// TIA Portal V20 program export: 3 tag tables, 23 data types, 15 data blocks, 37 code blocks (in call order from the OBs), 16 instance data blocks

VAR_GLOBAL   // PLC tag table "IO"
   "I_IN1_EXT+SGV" AT %I0.0 : Bool;   // communication spare (not used)
   "I_IN2_EXT+SGV" AT %I0.1 : Bool;   // communication spare (not used)
   "I_IN3_EXT+SGV" AT %I0.2 : Bool;   // communication spare (not used)
   "I_0E1+SGV" AT %I0.3 : Bool;   // air conditioner 1 scannerhousing visual measurement (1=ok)
   "I_0E2+SGX" AT %I0.4 : Bool;   // air conditioner scannerhousing x-ray measurement (1=ok)
   "I_0F1.1+SGV" AT %I0.5 : Bool;   // monitoring circuit breaker supply 24V ( -0F1.1)
   "I_0SH1+SSTR" AT %I0.6 : Bool;   // cooling fan / air conditioner off (cleaning filter)
   "I_14SB0+HMI" AT %I0.7 : Bool;   // emergency stop Goldeneye HMI
   "I_14SB1+HMI" AT %I1.0 : Bool;   // scanner release Goldeneye HMI
   "I_8S1.T_in" AT %I1.1 : Bool;   // adjustment top limit switch innermost position
   "I_8S2.T_out" AT %I1.2 : Bool;   // adjustment top limit switch outermost position
   "I_8S1.L_in" AT %I1.3 : Bool;   // adjustment left limit switch innermost position
   "I_8S2.L_out" AT %I1.4 : Bool;   // adjustment left limit switch outermost position
   "I_8S1.R_in" AT %I1.5 : Bool;   // adjustment right limit switch innermost position
   "I_8S2.R_out" AT %I1.6 : Bool;   // adjustment right limit switch outermost position
   "I_8S1.B_left" AT %I2.0 : Bool;   // adjustment scannerhousing limit switch left position
   "I_8S2.B_right" AT %I2.1 : Bool;   // adjustment scannerhousing limit switch right position
   "I_1BTR2+SGX" AT %I2.2 : Bool;   // light barrier in scannerhousing x-ray measurement
   "O_14VK1+SGV" AT %Q0.0 : Bool;   // safety loops scanner internal ok
   "O_14VK2+SGV" AT %Q0.1 : Bool;   // setting mode active
   "O_0VK1+SGV" AT %Q0.2 : Bool;   // scanner ready
   "O_0VK2+SGV" AT %Q0.3 : Bool;   // scanner error
   "O_0VK3+SGV" AT %Q0.4 : Bool;   // communication spare (not used)
   "O_0VK4+SGV" AT %Q0.5 : Bool;   // communication spare (not used)
   "O_0F1.1+SGV" AT %Q0.6 : Bool;   // acknowledge circuit breaker supply 24V
   "O_0KA0.1+SGV" AT %Q0.7 : Bool;   // air conditioner scannerhousing visual measurement off
   "O_0KA1+SGV" AT %Q1.1 : Bool;   // scanner status display
   "O_8M1.T_c" AT %Q1.2 : Bool;   // adjustment top close
   "O_8M1.T_o" AT %Q1.3 : Bool;   // adjustment top open
   "O_8M1.L_c" AT %Q1.4 : Bool;   // adjustment left close
   "O_8M1.L_o" AT %Q1.5 : Bool;   // adjustment left open
   "O_8M1.R_c" AT %Q1.6 : Bool;   // adjustment right close
   "O_8M1.R_o" AT %Q1.7 : Bool;   // adjustment right open
   "O_8M1.B_l" AT %Q2.1 : Bool;   // adjustment scannerhousing left
   "O_8M1.B_r" AT %Q2.2 : Bool;   // adjustment scannerhousing right
   "SI_NA_EXT+SGV" AT %I800.0 : Bool;   // emergency stop + area stop external
   "SI_14SB0/1+HMI" AT %I800.1 : Bool;   // emergency stop / scanner release Goldeneye HMI
   "SI_14SB1+SSTL" AT %I800.2 : Bool;   // setting mode scanner active
   "SI_14SB2+SSTL" AT %I800.3 : Bool;   // jog adjustment camera
   "SI_8U1+SGV" AT %I824.0 : Bool;   // adjustment linear drive monitoring
   "SI_14KA1+SGV" AT %I824.1 : Bool;   // area laser monitoring
   "SI_14KA2+SGV" AT %I824.2 : Bool;   // area adjustment monitoring
   "SI_14SS1.TL+SGV" AT %I808.0 : Bool;   // safety contact cover top left SGV
   "SI_14SS1.BL+SGV" AT %I808.1 : Bool;   // safety contact cover bottom left SGV
   "SI_14SS1.TR+SGV" AT %I808.2 : Bool;   // safety contact cover top right SGV
   "SI_14SS1.BR+SGV" AT %I808.3 : Bool;   // safety contact cover bottom right SGV
   "SI_14SS1.TL+SGX" AT %I816.0 : Bool;   // safety contact cover top left SGX
   "SI_14SS1.BL+SGX" AT %I816.1 : Bool;   // safety contact cover bottom left SGX
   "SI_14SS1.TR+SGX" AT %I816.2 : Bool;   // safety contact cover top right SGX
   "SI_14SS1.BR+SGX" AT %I816.3 : Bool;   // safety contact cover bottom right SGX
   "SO_14HV1+SSTL/R" AT %Q900.1 : Bool;   // setting mode scanner active
   "SO_14KA1+SGV" AT %Q900.2 : Bool;   // area laser on
   "SO_14KA2+SGV" AT %Q900.3 : Bool;   // area adjustment on
   "SO_ST.3HF+SGV" AT %Q908.0 : Bool;   // safety lamp laser on
   "SO_ST.5HF+SGV" AT %Q908.1 : Bool;   // safety lamp X-Ray on
   "SO_5AX1+SGX" AT %Q908.2 : Bool;   // area x-ray on
   "O_8KA1+SGV" AT %Q2.0 : Bool;   // adjustment linear drive reset (not used)
   "I_1BTR2+SGV" AT %I1.7 : Bool;   // light barrier in scannerhousing visual measurement
   "O_2YV1/2.B+SGV" AT %Q2.3 : Bool;   // blow-off valve SGV bottom
   "O_2YV1.L+SGV" AT %Q2.4 : Bool;   // blow-off valve SGV left
   "O_2YV1.R+SGV" AT %Q2.5 : Bool;   // blow-off valve SGV right
   "O_5YV1+SGX" AT %Q2.6 : Bool;   // blow-off valve SGX X-Ray
   "O_0KA0.2+SGV" AT %Q1.0 : Bool;   // air conditioner scannerhousing x-ray measurement off
   "SI_5AX1+SGX" AT %I824.3 : Bool;   // area x-ray monitoring
   O_spare27 AT %Q2.7 : Bool;   // output normal spare
   "I_0E1.1+SGV" AT %I2.3 : Bool;   // air conditioner 2 scannerhousing visual measurement (1=ok)
   I_spare24 AT %I2.4 : Bool;
   I_spare25 AT %I2.5 : Bool;
   I_spare26 AT %I2.6 : Bool;
   I_spare27 AT %I2.7 : Bool;
   SO_spare9083 AT %Q908.3 : Bool;
   SO_safetynew AT %Q900.0 : Bool;
   I_test AT %I5.0 : Bool;
END_VAR

VAR_GLOBAL   // PLC tag table "Standard-Variablentabelle"
   test0ibn AT %M0.4 : Bool;
   test1ibn AT %M0.5 : Bool;
   Tag_1 AT %M400.0 : Bool;
   Tag_2 AT %M400.1 : Bool;
   Tag_3 AT %M400.2 : Bool;
   Tag_4 AT %M2345.4 : Bool;
END_VAR
VAR_GLOBAL CONSTANT   // user constants
   USERDIAG_DEVICES_PER_SCREEN_UPPER_LIM : Int := 32;
   USERDIAG_SLOTS_PER_SCREEN_UPPER_LIM : Int := 31;
   USERDIAG_SLOTS_PER_DEVICE_UPPER_LIM : Int := 31;
   USERDIAG_DEVICES_PER_IO_SYSTEM_UPPER_LIM : Int := 128;
   USERDIAG_SLOTS_PER_PLC_UPPER_LIM : Int := 31;
END_VAR

VAR_GLOBAL   // PLC tag table "Standard"
   false AT %M0.0 : Bool;
   true AT %M0.1 : Bool;
   test0 AT %M0.2 : Bool;
   test1 AT %M0.3 : Bool;
   dummy AT %M0.7 : Bool;
   clockFlag10Hz AT %M1.0 : Bool;   // ClockFlag 0.1s
   clockFlag5Hz AT %M1.1 : Bool;   // ClockFlag 0.2s
   flash AT %M1.2 : Bool;   // ClockFlag 0.4s
   clockFlag2Hz AT %M1.3 : Bool;   // ClockFlag 0.5s
   blinker AT %M1.4 : Bool;   // ClockFlag 0.8s
   clockFlag1Hz AT %M1.5 : Bool;   // ClockFlag 1.0s
   "clockFlag0,625Hz" AT %M1.6 : Bool;   // ClockFlag 1.6s
   "clockFlag0,5Hz" AT %M1.7 : Bool;   // ClockFlag 2.0s
   cycleFlag AT %MB2 : Byte;
   cycleFlash AT %M2.0 : Bool;
   systemByte AT %MB3 : Byte;
   firstScan AT %M3.0 : Bool;   // cpu startup
   diagStatusUpdate AT %M3.1 : Bool;
   alwaysTRUE AT %M3.2 : Bool;
   alwaysFALSE AT %M3.3 : Bool;
   clockByte AT %MB1 : Byte;
   cycle AT %MD6 : Real;   // program cycle in ms
   "real" AT %MD10 : Real;
   "dWord" AT %MD18 : DWord;
   "dint" AT %MD14 : DInt;
   "int" AT %MW22 : Int;
   "word" AT %MW24 : Word;
   "byte" AT %MB26 : Byte;
   "bool" AT %M27.0 : Bool;
   systemClockByte AT %MB30 : Byte;
   clockTest AT %M0.6 : Bool;
   T0 AT %T0 : Timer;
   T1 AT %T1 : Timer;
   T2 AT %T2 : Timer;
   mem AT %M32.0 : LReal;
   T3 AT %T3 : Timer;
END_VAR

TYPE "TypeAxisRd"
   STRUCT
      TargetPos : DInt;   // target position [mm/10]
      CalibratePos : DInt;   // calibrated position [mm/10]
      RefPosToBoard : DInt;   // reference position to board [mm/10]
      SetCalibratePos : Bool;   // set calibrated position
      ManModeActive : Bool;   // manual mode active
      ManPlus : Bool;   // manual plus
      ManMinus : Bool;   // manual minus
      ManRefRun : Bool;   // manual reference run
   END_STRUCT;
END_TYPE

TYPE "TypeAxisSd"
   STRUCT
      ActualEncPos : DInt;   // actual encoder position [mm/10]
      ActualPos : DInt;   // actual position [mm/10]
      LimitSwitchMin : Bool;   // limit switch min active
      LimitSwitchMax : Bool;   // limit switch max active
      Err : Bool;   // error
      ErrEnc : Bool;   // error encoder
      PosOk : Bool;   // position ok
      Plus : Bool;   // moves plus
      Minus : Bool;   // moves minus
      refRun : Bool;   // reference running
      refOk : Bool;   // reference ok
      SetCalibratePosOk : Bool;   // set calibrated position ok
   END_STRUCT;
END_TYPE

TYPE "TypeCmd"
   STRUCT
      auto : Bool;   // automatic mode
      autoP : Bool;   // automatic plus
      autoM : Bool;   // automatic minus
      autoLift : Bool;   // automatic lift
      autoLower : Bool;   // automatic lower
      man : Bool;   // manual mode
      manP : Bool;   // manual plus
      manM : Bool;   // manual minus
      manLift : Bool;   // manual lift
      manLower : Bool;   // manual lower
      enable : Bool;   // release
      enPlus : Bool;   // release plus
      enMinus : Bool;   // release minus
      enLift : Bool;   // release lift
      enLower : Bool;   // release lower
      enAutoP : Bool;   // release automatic plus
      enAutoM : Bool;   // release automatic minus
      enAutoLift : Bool;   // release automatic lift
      enAutoLower : Bool;   // release automatic lower
      slow : Bool;
      lamp : Bool;   // indication lamp
      ack : Bool;   // fault acknowledge
      cycle : Bool;   // cycle start
      goToGpos : Bool;   // go to groundposition
      goToCpos : Bool;   // go to cm-position
      goToEpos : Bool;   // go to endpos
      goToWPos : Bool;   // go to wait/fly position
      inGpos : Bool;   // in groundposition
      inCpos : Bool;   // in cm-position
      inEpos : Bool;   // in endpos
      inWPos : Bool;   // in wait/fly position
      speed : Int;   // Desired speed raw in Hz or Upm
      tarSpeed : Real;   // target speed
      mmCycle : Real;   // milimeter per cycle
      gain : Real;   // gain
      ramp : Int;   // ramp
      startRamp : Int;   // start ramp
      stopRamp : Int;   // stop ramp
      gPos : Real;   // Desired value basic position [mm]
      cPos : Real;   // Desired value cm position [mm]
      ePos : Real;   // Desired value end position [mm]
      wPos : Real;   // Desired value wait/fly position [mm]
      tarMax : Real;   // target maximum
      tarMin : Real;   // target minimum
      target : Real;
      actual : Real;
   END_STRUCT;
END_TYPE

TYPE "TypeHeaderPcGld"
   STRUCT
      valid : Int;   // valid
      watchdog : Int;   // watchdog
      bit40 : Bool;
      ack : Bool;   // acknowledge
      bit42 : Bool;
      bit43 : Bool;
      bit44 : Bool;
      bit45 : Bool;
      bit46 : Bool;
      bit47 : Bool;
      word6 : Word;
      word8 : Word;
   END_STRUCT;
END_TYPE

TYPE "TypeHeaderPlc"
   STRUCT
      conActive : Bool;   // connection is established
      err : Bool;   // fault general
      errWd : Bool;   // fault watchdog
      errSd : Bool;   // fault send
      errRd : Bool;   // fault receive
      bit05 : Bool;
      bit06 : Bool;
      bit07 : Bool;
      sdBusy : Bool;   // new data is sending
      sdDone : Bool;   // new data sended
      rdBusy : Bool;   // new data is receiving
      rdDone : Bool;   // new data received
      sdOverload : Bool;   // new data could not be sent because the Cp overloaded
      statistic : Bool;   // statistic information are aviable
      bit16 : Bool;
      bit17 : Bool;
      sdState : Word;   // send state
      sdLastErrState : Word;   // send last fault state
      sdLenght : Int;   // send lenght [byte]
      sdCps : Int;   // send counter per second
      rdState : Word;   // receive state
      rdLastErrState : Word;   // receive last fault state
      rdLenght : Int;   // receive lenght [byte]
      rdCps : Int;   // receive counter per second
      in18 : Int;
   END_STRUCT;
END_TYPE

TYPE "TypeSensor"
   STRUCT
      sen : Bool;
      onDel : Bool;
      offDel : Bool;
      occ : Bool;
      occPe : Bool;
      occNe : Bool;
      off : Bool;
      full : Bool;
      free : Bool;
      empty : Bool;
      err : Bool;
      errOcc : Bool;   // fault sensor was to long occupied, maybe dirty or misaligned
      errFree : Bool;   // fault sensor was to long free, maybe dirty or misaligned
      errCycle : Bool;   // fault sensor plausibility check of cycles, after a certain amount(#errCycleVal) of trigger(#errCycleIn) the sensor had no rising or falling edge
      war : Bool;
      refMode : Bool;   // reference mode
      refRun : Bool;   // reference running
      onCntr : Real;   // counter for on delayed
      offCntr : Real;   // counter for off delayed
      occOnCntr : Real;   // on counter for occupied
      occOffCntr : Real;   // on counter for occupied
      val : Real;   // value from sensor, if ex. the sensor is read as a analog input
      occGap : Real;   // gap since last occupied
      "name" : WString[30];   // name, used for fault messages
      description : WString[90];   // description, used for fault messages
   END_STRUCT;
END_TYPE

TYPE "TypeVar"
   STRUCT
      "bool" { ExternalAccessible := 'False'; ExternalVisible := 'False'; ExternalWritable := 'False'} : Bool;
      "byte" { ExternalAccessible := 'False'; ExternalVisible := 'False'; ExternalWritable := 'False'} : Byte;
      "word" { ExternalAccessible := 'False'; ExternalVisible := 'False'; ExternalWritable := 'False'} : Word;
      "dword" { ExternalAccessible := 'False'; ExternalVisible := 'False'; ExternalWritable := 'False'} : DWord;
      "int" { ExternalAccessible := 'False'; ExternalVisible := 'False'; ExternalWritable := 'False'} : Int;
      "dint" { ExternalAccessible := 'False'; ExternalVisible := 'False'; ExternalWritable := 'False'} : DInt;
      "real" { ExternalAccessible := 'False'; ExternalVisible := 'False'; ExternalWritable := 'False'} : Real;
      s5time { ExternalAccessible := 'False'; ExternalVisible := 'False'; ExternalWritable := 'False'} : S5Time;
      "time" { ExternalAccessible := 'False'; ExternalVisible := 'False'; ExternalWritable := 'False'} : Time;
      hm1 { ExternalAccessible := 'False'; ExternalVisible := 'False'; ExternalWritable := 'False'} : Bool;
      hm2 { ExternalAccessible := 'False'; ExternalVisible := 'False'; ExternalWritable := 'False'} : Bool := false;
      hm3 { ExternalAccessible := 'False'; ExternalVisible := 'False'; ExternalWritable := 'False'} : Bool := false;
      hm4 { ExternalAccessible := 'False'; ExternalVisible := 'False'; ExternalWritable := 'False'} : Bool := false;
      hm5 { ExternalAccessible := 'False'; ExternalVisible := 'False'; ExternalWritable := 'False'} : Bool := false;
      hm6 { ExternalAccessible := 'False'; ExternalVisible := 'False'; ExternalWritable := 'False'} : Bool := false;
      hm7 { ExternalAccessible := 'False'; ExternalVisible := 'False'; ExternalWritable := 'False'} : Bool := false;
      hm8 { ExternalAccessible := 'False'; ExternalVisible := 'False'; ExternalWritable := 'False'} : Bool := false;
      hm9 { ExternalAccessible := 'False'; ExternalVisible := 'False'; ExternalWritable := 'False'} : Bool := false;
      hm10 { ExternalAccessible := 'False'; ExternalVisible := 'False'; ExternalWritable := 'False'} : Bool := false;
      hm11 { ExternalAccessible := 'False'; ExternalVisible := 'False'; ExternalWritable := 'False'} : Bool := false;
      hm12 { ExternalAccessible := 'False'; ExternalVisible := 'False'; ExternalWritable := 'False'} : Bool := false;
      hm13 { ExternalAccessible := 'False'; ExternalVisible := 'False'; ExternalWritable := 'False'} : Bool := false;
      hm14 { ExternalAccessible := 'False'; ExternalVisible := 'False'; ExternalWritable := 'False'} : Bool := false;
      hm15 { ExternalAccessible := 'False'; ExternalVisible := 'False'; ExternalWritable := 'False'} : Bool := false;
      hm16 { ExternalAccessible := 'False'; ExternalVisible := 'False'; ExternalWritable := 'False'} : Bool := false;
      fm1 { ExternalAccessible := 'False'; ExternalVisible := 'False'; ExternalWritable := 'False'} : Bool;
      fm2 { ExternalAccessible := 'False'; ExternalVisible := 'False'; ExternalWritable := 'False'} : Bool := false;
      fm3 { ExternalAccessible := 'False'; ExternalVisible := 'False'; ExternalWritable := 'False'} : Bool := false;
      fm4 { ExternalAccessible := 'False'; ExternalVisible := 'False'; ExternalWritable := 'False'} : Bool := false;
      fm5 { ExternalAccessible := 'False'; ExternalVisible := 'False'; ExternalWritable := 'False'} : Bool := false;
      fm6 { ExternalAccessible := 'False'; ExternalVisible := 'False'; ExternalWritable := 'False'} : Bool := false;
      fm7 { ExternalAccessible := 'False'; ExternalVisible := 'False'; ExternalWritable := 'False'} : Bool := false;
      fm8 { ExternalAccessible := 'False'; ExternalVisible := 'False'; ExternalWritable := 'False'} : Bool := false;
      fm9 { ExternalAccessible := 'False'; ExternalVisible := 'False'; ExternalWritable := 'False'} : Bool := false;
      fm10 { ExternalAccessible := 'False'; ExternalVisible := 'False'; ExternalWritable := 'False'} : Bool := false;
      fm11 { ExternalAccessible := 'False'; ExternalVisible := 'False'; ExternalWritable := 'False'} : Bool := false;
      fm12 { ExternalAccessible := 'False'; ExternalVisible := 'False'; ExternalWritable := 'False'} : Bool := false;
      fm13 { ExternalAccessible := 'False'; ExternalVisible := 'False'; ExternalWritable := 'False'} : Bool := false;
      fm14 { ExternalAccessible := 'False'; ExternalVisible := 'False'; ExternalWritable := 'False'} : Bool := false;
      fm15 { ExternalAccessible := 'False'; ExternalVisible := 'False'; ExternalWritable := 'False'} : Bool := false;
      fm16 { ExternalAccessible := 'False'; ExternalVisible := 'False'; ExternalWritable := 'False'} : Bool := false;
      bool1 { ExternalAccessible := 'False'; ExternalVisible := 'False'; ExternalWritable := 'False'} : Bool;
      bool2 { ExternalAccessible := 'False'; ExternalVisible := 'False'; ExternalWritable := 'False'} : Bool;
      bool3 { ExternalAccessible := 'False'; ExternalVisible := 'False'; ExternalWritable := 'False'} : Bool;
      bool4 { ExternalAccessible := 'False'; ExternalVisible := 'False'; ExternalWritable := 'False'} : Bool;
      bool5 { ExternalAccessible := 'False'; ExternalVisible := 'False'; ExternalWritable := 'False'} : Bool;
      bool6 { ExternalAccessible := 'False'; ExternalVisible := 'False'; ExternalWritable := 'False'} : Bool;
      bool7 { ExternalAccessible := 'False'; ExternalVisible := 'False'; ExternalWritable := 'False'} : Bool;
      bool8 { ExternalAccessible := 'False'; ExternalVisible := 'False'; ExternalWritable := 'False'} : Bool;
      bool9 { ExternalAccessible := 'False'; ExternalVisible := 'False'; ExternalWritable := 'False'} : Bool;
      bool10 { ExternalAccessible := 'False'; ExternalVisible := 'False'; ExternalWritable := 'False'} : Bool;
      bool11 { ExternalAccessible := 'False'; ExternalVisible := 'False'; ExternalWritable := 'False'} : Bool;
      bool12 { ExternalAccessible := 'False'; ExternalVisible := 'False'; ExternalWritable := 'False'} : Bool;
      bool13 { ExternalAccessible := 'False'; ExternalVisible := 'False'; ExternalWritable := 'False'} : Bool;
      bool14 { ExternalAccessible := 'False'; ExternalVisible := 'False'; ExternalWritable := 'False'} : Bool;
      bool15 { ExternalAccessible := 'False'; ExternalVisible := 'False'; ExternalWritable := 'False'} : Bool;
      bool16 { ExternalAccessible := 'False'; ExternalVisible := 'False'; ExternalWritable := 'False'} : Bool;
      int1 { ExternalAccessible := 'False'; ExternalVisible := 'False'; ExternalWritable := 'False'} : Int;
      int2 { ExternalAccessible := 'False'; ExternalVisible := 'False'; ExternalWritable := 'False'} : Int := 0;
      int3 { ExternalAccessible := 'False'; ExternalVisible := 'False'; ExternalWritable := 'False'} : Int := 0;
      int4 { ExternalAccessible := 'False'; ExternalVisible := 'False'; ExternalWritable := 'False'} : Int := 0;
      int5 { ExternalAccessible := 'False'; ExternalVisible := 'False'; ExternalWritable := 'False'} : Int := 0;
      int6 { ExternalAccessible := 'False'; ExternalVisible := 'False'; ExternalWritable := 'False'} : Int := 0;
      int7 { ExternalAccessible := 'False'; ExternalVisible := 'False'; ExternalWritable := 'False'} : Int := 0;
      int8 { ExternalAccessible := 'False'; ExternalVisible := 'False'; ExternalWritable := 'False'} : Int := 0;
      int9 { ExternalAccessible := 'False'; ExternalVisible := 'False'; ExternalWritable := 'False'} : Int := 0;
      int10 { ExternalAccessible := 'False'; ExternalVisible := 'False'; ExternalWritable := 'False'} : Int := 0;
      word1 { ExternalAccessible := 'False'; ExternalVisible := 'False'; ExternalWritable := 'False'} : Word;
      word2 { ExternalAccessible := 'False'; ExternalVisible := 'False'; ExternalWritable := 'False'} : Word := 16#0;
      word3 { ExternalAccessible := 'False'; ExternalVisible := 'False'; ExternalWritable := 'False'} : Word := 16#0;
      word4 { ExternalAccessible := 'False'; ExternalVisible := 'False'; ExternalWritable := 'False'} : Word := 16#0;
      word5 { ExternalAccessible := 'False'; ExternalVisible := 'False'; ExternalWritable := 'False'} : Word := 16#0;
      word6 { ExternalAccessible := 'False'; ExternalVisible := 'False'; ExternalWritable := 'False'} : Word := 16#0;
      word7 { ExternalAccessible := 'False'; ExternalVisible := 'False'; ExternalWritable := 'False'} : Word := 16#0;
      word8 { ExternalAccessible := 'False'; ExternalVisible := 'False'; ExternalWritable := 'False'} : Word := 16#0;
      word9 { ExternalAccessible := 'False'; ExternalVisible := 'False'; ExternalWritable := 'False'} : Word := 16#0;
      word10 { ExternalAccessible := 'False'; ExternalVisible := 'False'; ExternalWritable := 'False'} : Word := 16#0;
      real1 { ExternalAccessible := 'False'; ExternalVisible := 'False'; ExternalWritable := 'False'} : Real;
      real2 { ExternalAccessible := 'False'; ExternalVisible := 'False'; ExternalWritable := 'False'} : Real := 0.0;
      real3 { ExternalAccessible := 'False'; ExternalVisible := 'False'; ExternalWritable := 'False'} : Real := 0.0;
      real4 { ExternalAccessible := 'False'; ExternalVisible := 'False'; ExternalWritable := 'False'} : Real := 0.0;
      real5 { ExternalAccessible := 'False'; ExternalVisible := 'False'; ExternalWritable := 'False'} : Real := 0.0;
      real6 { ExternalAccessible := 'False'; ExternalVisible := 'False'; ExternalWritable := 'False'} : Real := 0.0;
      real7 { ExternalAccessible := 'False'; ExternalVisible := 'False'; ExternalWritable := 'False'} : Real := 0.0;
      real8 { ExternalAccessible := 'False'; ExternalVisible := 'False'; ExternalWritable := 'False'} : Real := 0.0;
      real9 { ExternalAccessible := 'False'; ExternalVisible := 'False'; ExternalWritable := 'False'} : Real := 0.0;
      real10 { ExternalAccessible := 'False'; ExternalVisible := 'False'; ExternalWritable := 'False'} : Real := 0.0;
   END_STRUCT;
END_TYPE

TYPE "UserDiag_typeActIOSystem"
TITLE = UserDiag_typeActIOSystem
   STRUCT
      actIOSystemNumber : Int := 1;   // Number of actual selected IO-system/DP-Mastersystem
      actIODeviceNumbers : Array[1.."USERDIAG_DEVICES_PER_SCREEN_UPPER_LIM"] of UInt;   // Device numbers/profibus addresses of actual selected IO-System/DP-Mastersystem
      actIODeviceState : Array[1.."USERDIAG_DEVICES_PER_SCREEN_UPPER_LIM"] of USInt;   // State of devices/slaves in actual selected IO-System/DP-Mastersystem
      actDeviceSlotsUsed : Array[0.."USERDIAG_SLOTS_PER_SCREEN_UPPER_LIM"] of Bool;   // Used slots of actual selected device/slave
      actDeviceSlotsState : Array[0.."USERDIAG_SLOTS_PER_SCREEN_UPPER_LIM"] of USInt;   // States of actual selected device/slave
   END_STRUCT;
END_TYPE

TYPE "UserDiag_typeDevice"
TITLE = UserDiag_typeDevice
   STRUCT
      hardwareId { ExternalAccessible := 'False'; ExternalVisible := 'False'; ExternalWritable := 'False'} : HW_DEVICE := 16#0000;   // Hardware identifier of the device/slave
      number { ExternalAccessible := 'False'; ExternalVisible := 'False'; ExternalWritable := 'False'} : UInt := 0;   // Profinet device number/Profibus address of the slave
      "name" { ExternalAccessible := 'False'; ExternalVisible := 'False'; ExternalWritable := 'False'} : String[50];   // Name of the device/slave
      ipAddress { ExternalAccessible := 'False'; ExternalVisible := 'False'; ExternalWritable := 'False'; S7_SetPoint := 'True'} : IP_V4;   // IP address of the device
      state { ExternalAccessible := 'False'; ExternalVisible := 'False'; ExternalWritable := 'False'} : USInt := 0;   // Status of the device/slave. 1:ok; 2:faulty, 3:lost connection, 4:disabled, 5:problem, 12:was faulty, 13:was lost, 14:was disabled, 15:problem gone
      exists { ExternalAccessible := 'False'; ExternalVisible := 'False'; ExternalWritable := 'False'} : Bool := FALSE;   // TRUE: Device/slave is existing
      configured { ExternalAccessible := 'False'; ExternalVisible := 'False'; ExternalWritable := 'False'} : Bool := FALSE;   // TRUE: Device/slave is configured
      faulty { ExternalAccessible := 'False'; ExternalVisible := 'False'; ExternalWritable := 'False'} : Bool := FALSE;   // TRUE: Device/slave is faulty
      problem { ExternalAccessible := 'False'; ExternalVisible := 'False'; ExternalWritable := 'False'} : Bool := FALSE;   // TRUE: Device/slave has a problem
      disabled { ExternalAccessible := 'False'; ExternalVisible := 'False'; ExternalWritable := 'False'} : Bool := FALSE;   // TRUE: Device/slave is disabled
      error { ExternalAccessible := 'False'; ExternalVisible := 'False'; ExternalWritable := 'False'} : Bool := FALSE;   // TRUE: Error in device/slave
      nextDevice { ExternalAccessible := 'False'; ExternalVisible := 'False'; ExternalWritable := 'False'} : Int;   // device number of next device
      actualConfiguredSlots { ExternalAccessible := 'False'; ExternalVisible := 'False'; ExternalWritable := 'False'} : Int := 0;   // Number of configured slots in the device/slave
      slots { ExternalAccessible := 'False'; ExternalVisible := 'False'; ExternalWritable := 'False'; S7_SetPoint := 'True'} : Array[0.."USERDIAG_SLOTS_PER_DEVICE_UPPER_LIM"] of "UserDiag_typeSlot";   // Slot information of a device/slave
   END_STRUCT;
END_TYPE

TYPE "UserDiag_typeDiagnostics"
TITLE = UserDiag_typeDiagnostics
   STRUCT
      subfunctionStatus : Word := 16#0000;   // Block status or error information
      instructionError : Int := 0;   // Indicates in which system function the error occurred. 1:DeviceStates PN; 2=GetName PN; 3:ModuleStates PN; 4:DeviceStates DP; 5:GetName DP; 6:ModuleStates DP
      errorIndex : Int := 0;   // The last index of the respective loop, if an error occures (relevant for IOSystemCheck FB)
   END_STRUCT;
END_TYPE

TYPE "UserDiag_typeIOSystem"
TITLE = UserDiag_typeIOSystem
   STRUCT
      hardwareId { ExternalAccessible := 'False'; ExternalVisible := 'False'; ExternalWritable := 'False'} : HW_IOSYSTEM := 16#0000;   // Hardware identifier of the IO-System/DP-Mastersystem
      number { ExternalAccessible := 'False'; ExternalVisible := 'False'; ExternalWritable := 'False'} : UInt := 0;   // IO-System/DP-Mastersystem number
      error { ExternalAccessible := 'False'; ExternalVisible := 'False'; ExternalWritable := 'False'} : Bool := FALSE;   // TRUE: Error in IO-System/DP-Mastersystem
      firstDevice { ExternalAccessible := 'False'; ExternalVisible := 'False'; ExternalWritable := 'False'} : Int := 0;   // device number (index) of first device in IO System
      lastDevice { ExternalAccessible := 'False'; ExternalVisible := 'False'; ExternalWritable := 'False'} : Int := 0;   // device number (index) of last device IO System
      actualConfiguredDevices { ExternalAccessible := 'False'; ExternalVisible := 'False'; ExternalWritable := 'False'} : Int := 0;   // Number of configured devices/slaves in IO-System/DP-Mastersystem
      devices { ExternalAccessible := 'False'; ExternalVisible := 'False'; ExternalWritable := 'False'; S7_SetPoint := 'True'} : Array[1.."USERDIAG_DEVICES_PER_IO_SYSTEM_UPPER_LIM"] of "UserDiag_typeDevice";   // Device/Slave information
   END_STRUCT;
END_TYPE

TYPE "UserDiag_typePLC"
TITLE = UserDiag_typePLC
   STRUCT
      hardwareId { ExternalAccessible := 'False'; ExternalVisible := 'False'; ExternalWritable := 'False'} : HW_DEVICE := 16#0000;   // Hardware identifier of the PLC
      error { ExternalAccessible := 'False'; ExternalVisible := 'False'; ExternalWritable := 'False'} : Bool := FALSE;   // TRUE: Error in PLC
      errorLedActive { ExternalAccessible := 'False'; ExternalVisible := 'False'; ExternalWritable := 'False'} : Bool := FALSE;   // TRUE: PLC led signals an error
      actualConfiguredSlots { ExternalAccessible := 'False'; ExternalVisible := 'False'; ExternalWritable := 'False'} : Int := 0;   // Number of configured local slots at PLC
      slots { ExternalAccessible := 'False'; ExternalVisible := 'False'; ExternalWritable := 'False'; S7_SetPoint := 'True'} : Array[0.."USERDIAG_SLOTS_PER_PLC_UPPER_LIM"] of "UserDiag_typeSlot";   // Information of the PLC slots; index = slotnumber; PLC always at slot 1
   END_STRUCT;
END_TYPE

TYPE "UserDiag_typeSlot"
TITLE = UserDiag_typeSlot
   STRUCT
      hardwareId { ExternalAccessible := 'False'; ExternalVisible := 'False'; ExternalWritable := 'False'} : HW_IO := 16#0000;   // Hardware identifier of the module which is inserted in the slot
      state { ExternalAccessible := 'False'; ExternalVisible := 'False'; ExternalWritable := 'False'} : USInt := 0;   // Status of the device/slave. 1:ok; 2:faulty, 3:lost connection, 4:disabled, 5:problem, 12:was faulty, 13:was lost, 14:was disabled, 15:problem gone
      exists { ExternalAccessible := 'False'; ExternalVisible := 'False'; ExternalWritable := 'False'} : Bool := FALSE;   // TRUE: Modul is existing
      configured { ExternalAccessible := 'False'; ExternalVisible := 'False'; ExternalWritable := 'False'} : Bool := FALSE;   // TRUE: Modul is configured
      faulty { ExternalAccessible := 'False'; ExternalVisible := 'False'; ExternalWritable := 'False'} : Bool := FALSE;   // TRUE: Modul is faulty
      problem { ExternalAccessible := 'False'; ExternalVisible := 'False'; ExternalWritable := 'False'} : Bool := FALSE;   // TRUE: Modul has a problem
      disabled { ExternalAccessible := 'False'; ExternalVisible := 'False'; ExternalWritable := 'False'} : Bool := FALSE;   // TRUE: Modul is disabled
      error { ExternalAccessible := 'False'; ExternalVisible := 'False'; ExternalWritable := 'False'} : Bool := FALSE;   // TRUE: Error in module which is inserted in the slot
   END_STRUCT;
END_TYPE

TYPE "TypeLinmotRd"
   STRUCT
      StatVar : Struct   // State Var
         SubState : Byte;   // main state
         MainState : Byte;   // sub state
      END_STRUCT;
      StatWord : Struct   // Status Word
         OperationEnabled : Bool;   // 1 = State Nr 8 or higher (copied to drive EN LED )
         SwitchOnActive : Bool;   // 1 = Control Word Bit 0
         EnableOperation : Bool;   // 1 = Control Word Bit 3
         Error : Bool;   // 1 = Error
         VoltageEnable : Bool;   // 1 = Control Word Bit 1
         QuickStop : Bool;   // 1 = Control Word Bit 2
         SwitchOnLocked : Bool;   // 1= Release with 0 of Control word bit 0 (Switch On)
         Warning : Bool;   // 1 = One or more bits in the Warn Word are set
         EventHandlerActive : Bool;   // Event Handler setup
         SpecialMotionActive : Bool;   // Special motion commands (Homing, ..) runs
         InTargetPosition : Bool;   // Actual position after motion in window
         Homed : Bool;   // Position sensor system valid
         FatalError : Bool;   // A fatal error can not be acknowledged!
         MotionActive : Bool;   // Setpoint generation (VAI, curve) active
         RangeIndicator1 : Bool;   // Defined UPID is in Range 1
         RangeIndicator2 : Bool;   // Defined UPID is in Range 2
      END_STRUCT;
      WarnWord : Struct   // Warning Word
         MotorHotSensor : Bool;
         MotorShortTimerOverload : Bool;
         MotorSupplyVoltageLow : Bool;
         MotorSupplyVoltageHigh : Bool;
         PositionLagAlways : Bool;
         Res5 : Bool;
         DriveHot : Bool;
         MotorNotHomed : Bool;
         PTC_Sensor1Hot : Bool;
         PTC_Sensor2Hot : Bool;
         Res10 : Bool;
         Res11 : Bool;
         Res12 : Bool;
         Res13 : Bool;
         InterfaceWarnFlag : Bool;
         ApplicationWarnFlag : Bool;
      END_STRUCT;
      Tarpos : DInt;   // target position
      Actpos : DInt;   // actual position
      TarCurrent : DInt;   // target current
      CfgStatWord : Int;   // config status word
      CfgId : Int;   // config index response
      CfgVal : DInt;   // config value response
   END_STRUCT;
END_TYPE

TYPE "TypeLinmotSd"
   STRUCT
      Ctrl : Struct   // control word
         SwitchOn : Bool;   // 0 = A-Stop, -> Current = 0, power switches disabled
         VoltageEnable : Bool;   // 0 = Power switches disabled without microcontroller action
         QuickStop : Bool;   // 0 = Quick Stop -> Current = 0 -> H-Bridges disabled
         EnableOperation : Bool;   // Position controller active Motion Commands enabled
         Abort : Bool;   // 0 = Quick Stop position control rests active, motion
         Freeze : Bool;   // 0 = Quick Stop position control rests active, Target position
         GoToPosition : Bool;   // 1 = Go to fixed parameterized Position. Wait for release of signal
         ErrorAcknoledge : Bool;   // 1 = Rising edge of signal acknowledges error
         JogMovePlus : Bool;   // 1 = Jog Move +
         JogMoveMinus : Bool;   // 1 = Jog Move -
         SpecialMove : Bool;   // 1 = Special Mode
         Home : Bool;   // 1 = At startup bit 11 Status word is cleared, until procedure
         ClearanceCheck : Bool;   // 1 = Enable Clearance Check Movement
         GoToInitialPosition : Bool;   // 1 = Rising edge will start go to initial position
         Linearizing : Bool;   // Reserved
         PhaseSearch : Bool;   // 1 = Enable Phase Search Movements
      END_STRUCT;
      McHd : Struct   // motion command header
         CC0 : Bool;   // Command Count bit 0
         CC1 : Bool;   // Command Count bit 1
         CC2 : Bool;   // Command Count bit 2
         CC3 : Bool;   // Command Count bit 3
         SubID0 : Bool;   // Sub ID bit 0
         SubID1 : Bool;   // Sub ID bit 1
         SubID2 : Bool;   // Sub ID bit 2
         SubID3 : Bool;   // Sub ID bit 3
         MasterID : Byte;   // Master ID
      END_STRUCT;
      McPar1 : DInt;   // motion command parameter 1
      McPar2 : DInt;   // motion command parameter 2
      McPar3 : DInt;   // motion command parameter 3
      McPar4 : DInt;   // motion command parameter 4
      McPar5 : DInt;   // motion command parameter 5
      CgfHd : Int;   // Config Header
      CfgId : Int;   // Config Index
      CfgVal : DInt;   // Config Value
   END_STRUCT;
END_TYPE

TYPE "TypeIOLinkParam"
   STRUCT
      Info { ExternalAccessible := 'False'; ExternalVisible := 'False'; ExternalWritable := 'False'} : String[16];
      Index { ExternalAccessible := 'False'; ExternalVisible := 'False'; ExternalWritable := 'False'} : Int;
      Subindex { ExternalAccessible := 'False'; ExternalVisible := 'False'; ExternalWritable := 'False'} : Int;
      Len { ExternalAccessible := 'False'; ExternalVisible := 'False'; ExternalWritable := 'False'} : Int;
      Value { ExternalAccessible := 'False'; ExternalVisible := 'False'; ExternalWritable := 'False'; S7_SetPoint := 'True'} : "TypeIOLinkParamData";
      Send { ExternalAccessible := 'False'; ExternalVisible := 'False'; ExternalWritable := 'False'} : "TypeIOLinkParamSend";
      Rec { ExternalAccessible := 'False'; ExternalVisible := 'False'; ExternalWritable := 'False'} : "TypeIOLinkParamRec";
   END_STRUCT;
END_TYPE

TYPE "TypeIOLinkParamArray"
   STRUCT
      Param { ExternalAccessible := 'False'; ExternalVisible := 'False'; ExternalWritable := 'False'} : Array[0..9] of "TypeIOLinkParam";
   END_STRUCT;
END_TYPE

TYPE "TypeIOLinkParamData"
   STRUCT
      data { ExternalAccessible := 'False'; ExternalVisible := 'False'; ExternalWritable := 'False'} : Array[0..31] of Byte;
   END_STRUCT;
END_TYPE

TYPE "TypeIOLinkParamRec"
   STRUCT
      Count { ExternalAccessible := 'False'; ExternalVisible := 'False'; ExternalWritable := 'False'} : Int;
      Rec { ExternalAccessible := 'False'; ExternalVisible := 'False'; ExternalWritable := 'False'} : Int;
      Info { ExternalAccessible := 'False'; ExternalVisible := 'False'; ExternalWritable := 'False'} : String[16];
      State { ExternalAccessible := 'False'; ExternalVisible := 'False'; ExternalWritable := 'False'} : Word;
   END_STRUCT;
END_TYPE

TYPE "TypeIOLinkParamSend"
   STRUCT
      Count { ExternalAccessible := 'False'; ExternalVisible := 'False'; ExternalWritable := 'False'} : Int;
      Send { ExternalAccessible := 'False'; ExternalVisible := 'False'; ExternalWritable := 'False'} : Int;
      Info { ExternalAccessible := 'False'; ExternalVisible := 'False'; ExternalWritable := 'False'} : String[16];
      State { ExternalAccessible := 'False'; ExternalVisible := 'False'; ExternalWritable := 'False'} : Word;
   END_STRUCT;
END_TYPE

TYPE "TypeBaluffBUS007xRd"
   STRUCT
      Measure : Int;   // Actual measured value 300...3500 1/10mm (-1= Read error)
      Scale : SInt;   // Scale -1 = 1/10mm
      SCC1 : Bool;   // Signal output 1 (1= Occ)
      res1 : Bool;
      res2 : Bool;
      res3 : Bool;
      res4 : Bool;
      res5 : Bool;
      res6 : Bool;
      res7 : Bool;
   END_STRUCT;
END_TYPE

TYPE "TypeWenglorP3PC301Rd"
   STRUCT
      Measure : DInt;   // Actual measured value 60.000...66000µm (-1= Read error)
      Scale : SInt;   // Scale -6 = µm
      SCC1 : Bool;   // Signal output 1 (1= Occ)
      SCC2 : Bool;   // Signal output 2 (1= Occ)
      Err : Bool;   // Signal sensor error (1= Error)
      Warn : Bool;   // Signal sensor warning(1= warning)
      Warn1 : Bool;   // Indication Error / Warning (1= true)
      Warn2 : Bool;   // Indication Error / Warning (1= true)
      Warn3 : Bool;   // Indication Error / Warning (1= true)
      Warn4 : Bool;   // Indication Error / Warning (1= true)
   END_STRUCT;
END_TYPE

TYPE "TypeWenglorP3PC301Sd"
   STRUCT
      LaserOff : Bool;   // Laser off (1=Off)
      Localization : Bool;   // Localization (1=On)
      res2 : Bool;
      SCC1TeachIn : Bool;   // Start Teach SCC1
      SCC2TeachIn : Bool;   // Start Teach SCC2
      res5 : Bool;
      res6 : Bool;
      res7 : Bool;
   END_STRUCT;
END_TYPE

DATA_BLOCK "SiCom"   // DB48
{ S7_Optimized_Access := 'TRUE' }
// stored: AutoNumber false, MemoryReserve 100
   VAR
      Ack : Bool;   // reset faults general
      LampTest : Struct   // lamp test
         SettingMode : Bool;   // setting mode
         LaserOn : Bool;   // laser on
         XrayOn : Bool;   // xray on
      END_STRUCT;
      Blinker : Bool;   // blinker
      Flash : Bool;   // flash
      SafetyTest : Bool;   // safety test
      AreaLaserOn : Bool;   // area laser on
      AreaAdjustmentOn : Bool;   // area adjustment on
      AreaXrayOn : Bool;   // area X-Ray on
      ResetSafetyDevice : Bool;   // reset safety devices
   END_VAR
BEGIN
END_DATA_BLOCK

DATA_BLOCK "ComErr"   // DB363
{ S7_Optimized_Access := 'FALSE' }
// stored: AutoNumber false
   VAR
      Plc : "TypeHeaderPlc";   // Header Plc
      Pc : "TypeHeaderPcGld";   // Header Pc
      Err : Array[2000..2599] of Bool;
   END_VAR
BEGIN
END_DATA_BLOCK

DATA_BLOCK "ComErrText"   // DB370
{ S7_Optimized_Access := 'TRUE' }
// stored: AutoNumber false, MemoryReserve 0
   VAR
      Plc : "TypeHeaderPlc";   // Header Plc
      Rd : Struct
         Pc : Struct
            watchdog : Bool;
            bit01 : Bool;
            bit02 : Bool;
            bit03 : Bool;
            bit04 : Bool;
            bit05 : Bool;
            bit06 : Bool;
            ack : Bool;
            word2 : Word;
            word4 : Word;
            word6 : Word;
            word8 : Word;
         END_STRUCT;
         language { S7_SetPoint := 'True'} : Array[1..3] of WString[2];   // language for alarm text [ISO639-1] (not used)
      END_STRUCT;
      Sd : Struct
         Pc : Struct
            watchdog : Bool;
            bit01 : Bool;
            bit02 : Bool;
            bit03 : Bool;
            bit04 : Bool;
            bit05 : Bool;
            bit06 : Bool;
            ack : Bool;
            word2 : Word;
            word4 : Word;
            word6 : Word;
            word8 : Word;
         END_STRUCT;
         language { S7_SetPoint := 'True'} : Array[1..3] of WString[2];   // language for alarm text [ISO639-1]
         errAct { ExternalAccessible := 'False'; ExternalVisible := 'False'; ExternalWritable := 'False'} : Array[1..20] of Struct   // alarm text for the most prior actual alarms on the plc
            idProd : UInt;   // producer Id (for Plc: 0=Program_Alarm, 4=SysDiag, 5=MotionControl, 6=Security, 8=GRAPH, 9=ProDiag)
            id : UInt;   // alarm Id (nr of alarm in the plc)
            prio : UInt;   // 0 .. 16 (0-1=info, 2=safety, 3=warning, 4-16=fault)
            timeStamp : LDT;   // UTC time [8Byte, LDT#2008-10-25-08:12:34.567]
            alarm : Array[1..3] of WString[254];   // alarm text
            info : Array[1..3] of WString[254];   // info text, cause of the alarm
            remedy : Array[1..3] of WString[254];   // remedy text, suggestion how to fix the fault
         END_STRUCT;
         errList : Struct   // alarm text to fill error list on Pc
            idProd : UInt;   // producer Id (for Plc: 0=Program_Alarm, 4=SysDiag, 5=MotionControl, 6=Security, 8=GRAPH, 9=ProDiag)
            id : UInt;   // alarm Id (Nr in error List)
            prio : UInt;   // 0 .. 16 (0-1=info, 2=safety, 3=warning, 4-16=fault)
            timeStamp : LDT;   // UTC time [8Byte, LDT#2008-10-25-08:12:34.567]
            alarm : Array[1..3] of WString[254];   // alarm text
            info : Array[1..3] of WString[254];   // info text, cause of the alarm
            remedy : Array[1..3] of WString[254];   // remedy text, suggestion how to fix the fault
         END_STRUCT;
      END_STRUCT;
   END_VAR
BEGIN
END_DATA_BLOCK

DATA_BLOCK "ComRd"   // DB361
{ S7_Optimized_Access := 'FALSE' }
// stored: AutoNumber false
   VAR
      Plc : "TypeHeaderPlc";   // Header Plc
      Pc : "TypeHeaderPcGld";   // Header Pc
      Data : Struct
         Config : Struct   // config
            "version" : Int;   // version info
            active : Bool;   // config active (Test Output not active)
            adjScannerActive : Bool;   // adjustment scanner housing active
            adjTopActive : Bool;   // adjustment metering bar top active
            adjLeftActive : Bool;   // adjustment metering bar left active
            adjRightActive : Bool;   // adjustment metering bar right active
            adjTopLinMotActive : Bool;   // adjustment metering bar top active - linear drive
            adjLeftLinMotActive : Bool;   // adjustment metering bar left active - linear drive
            adjRightLinMotActive : Bool;   // adjustment metering bar right active - linear drive
            xrayActive : Bool;   // xray active
            adjLaserTopLeftStepMotActive : Bool;   // adjustment laser top left active - step motor
            adjLaserTopRightStepMotActive : Bool;   // adjustment laser top right active - step motor
            adjLaserLeftTopStepMotActive : Bool;   // adjustment laser left top active - step motor
            adjLaserLeftBottomStepMotActive : Bool;   // adjustment laser left bottom active - step motor
            adjLaserRightTopStepMotActive : Bool;   // adjustment laser right top active - step motor
            adjLaserRightBottomStepMotActive : Bool;   // adjustment laser right bottom active - step motor
            modeBoardPassing : Int;   // 1=left / 2=rigth / 3=middle
            modeDimension : Int;   // 1=fixed / 2=random width / 3=random thickness / 4=random width + thickness
            modeRandomAdj : Int;   // 1=with sensor / 2=with external data
            spare40 : Int;   // spare
            spare42 : Int;   // spare
            enc1Factor : Int;   // encoder infeed factor
            spare46 : Int;   // spare
            spare48 : Int;   // spare
            enc1QuadEvalActive : Bool;   // encoder infeed - quadruple evaluation active
            spare501 : Bool;   // spare
            spare502 : Bool;   // spare
         END_STRUCT;
         control : Struct   // control
            spare1 : Bool;
            spare2 : Bool;
         END_STRUCT;
         safety : Struct   // safety
            AreaLaserOn : Bool;   // area laser on
            AreaAdjustmentOn : Bool;   // area adjustment on
            AreaXrayOn : Bool;   // area X-Ray on
            ResetSafetyDevice : Bool;   // reset safety device
         END_STRUCT;
         status : Struct   // status
            Auto : Bool;   // automatic mode scanner
            StopFeeding : Bool;   // stop feeding scanner (error active)
         END_STRUCT;
         batch : Struct   // batch info
            MinWidth : DInt;   // min width [mm/10]
            MaxWidth : DInt;   // max width [mm/10]
            MinThickness : DInt;   // min thickness [mm/10]
            MaxThickness : DInt;   // max thickness [mm/10]
         END_STRUCT;
         Scanner : "TypeAxisRd";   // adjustment scanner
         Top : "TypeAxisRd";   // adjustment top
         Left : "TypeAxisRd";   // adjustment left
         Right : "TypeAxisRd";   // adjustment right
         Measure : Struct   // measuring sensor for random width/thickness
            SetCalibratePosTop : Bool;   // set calibrated position for sensor top
            SetCalibratePosLeft : Bool;   // set calibrated position for sensor left
            SetCalibratePosRight : Bool;   // set calibrated position for sensor right
         END_STRUCT;
         TestOutput : Struct   // test output
            Active : Bool;   // test output active
            "Q0.0" : Bool;
            "Q0.1" : Bool;
            "Q0.2" : Bool;
            "Q0.3" : Bool;
            "Q0.4" : Bool;
            "Q0.5" : Bool;
            "Q0.6" : Bool;
            "Q0.7" : Bool;
            "Q1.0" : Bool;
            "Q1.1" : Bool;
            "Q2.0" : Bool;
            "Q2.3" : Bool;
            "Q2.4" : Bool;
            "Q2.5" : Bool;
            "Q2.6" : Bool;
            "Q900.1" : Bool;
            "Q908.0" : Bool;
            "Q908.1" : Bool;
         END_STRUCT;
         res : Array[1..200] of Byte;
      END_STRUCT;
   END_VAR
BEGIN
END_DATA_BLOCK

DATA_BLOCK "ComSd"   // DB362
{ S7_Optimized_Access := 'FALSE' }
// stored: AutoNumber false
   VAR
      Plc : "TypeHeaderPlc";   // Header Plc
      Pc : "TypeHeaderPcGld";   // Header Pc
      Data : Struct
         config : Struct   // config
            "Version" : Int;   // version info
            spare2 : Int;
            spare3 : Int;
            spare4 : Int;
         END_STRUCT;
         control : Struct   // control
            spare : Bool;
         END_STRUCT;
         safety : Struct   // safety
            AreaLaserOn : Bool;   // area laser on
            AreaAdjustmentOn : Bool;   // area adjustment on
            AreaXrayOn : Bool;   // area X-Ray on
            spare : Bool;
         END_STRUCT;
         status : Struct   // status
            ready : Bool;   // plc ready
            err : Bool;   // plc error
         END_STRUCT;
         Scanner : "TypeAxisSd";   // adjustment scanner
         Top : "TypeAxisSd";   // adjustment top
         Left : "TypeAxisSd";   // adjustment left
         Right : "TypeAxisSd";   // adjustment right
         Measure : Struct   // measuring sensor for random width/thickness
            ActValueTop : DInt;   // actual value [mm/10]
            ActValueLeft : DInt;   // actual value [mm/10]
            ActValueRight : DInt;   // actual value [mm/10]
            Thickness : DInt;   // thickness [mm/10]
            Width : DInt;   // width [mm/10]
            SetCalibratePosTopOk : Bool;   // set calibrated position for sensor top ok
            SetCalibratePosLeftOk : Bool;   // set calibrated position for sensor left ok
            SetCalibratePosRightOk : Bool;   // set calibrated position for sensor right ok
         END_STRUCT;
         PlcInputNormal : Struct   // plc Input normal
            "I0.0" : Bool;
            "I0.1" : Bool;
            "I0.2" : Bool;
            "I0.3" : Bool;
            "I0.4" : Bool;
            "I0.5" : Bool;
            "I0.6" : Bool;
            "I0.7" : Bool;
            "I1.0" : Bool;
            "I1.1" : Bool;
            "I1.2" : Bool;
            "I1.3" : Bool;
            "I1.4" : Bool;
            "I1.5" : Bool;
            "I1.6" : Bool;
            "I1.7" : Bool;
            "I2.0" : Bool;
            "I2.1" : Bool;
            "I2.2" : Bool;
            "I2.3" : Bool;
            "I2.4" : Bool;
            "I2.5" : Bool;
            "I2.6" : Bool;
            "I2.7" : Bool;
         END_STRUCT;
         PlcInputSafety : Struct   // plc Input safety
            "I800.0" : Bool;
            "I800.1" : Bool;
            "I800.2" : Bool;
            "I800.3" : Bool;
            "I808.0" : Bool;
            "I808.1" : Bool;
            "I808.2" : Bool;
            "I808.3" : Bool;
            "I816.0" : Bool;
            "I816.1" : Bool;
            "I816.2" : Bool;
            "I816.3" : Bool;
            "I824.0" : Bool;
            "I824.1" : Bool;
            "I824.2" : Bool;
            "I824.3" : Bool;
         END_STRUCT;
         PlcOutputNormal : Struct   // plc output normal
            "Q0.0" : Bool;
            "Q0.1" : Bool;
            "Q0.2" : Bool;
            "Q0.3" : Bool;
            "Q0.4" : Bool;
            "Q0.5" : Bool;
            "Q0.6" : Bool;
            "Q0.7" : Bool;
            "Q1.0" : Bool;
            "Q1.1" : Bool;
            "Q1.2" : Bool;
            "Q1.3" : Bool;
            "Q1.4" : Bool;
            "Q1.5" : Bool;
            "Q1.6" : Bool;
            "Q1.7" : Bool;
            "Q2.0" : Bool;
            "Q2.1" : Bool;
            "Q2.2" : Bool;
            "Q2.3" : Bool;
            "Q2.4" : Bool;
            "Q2.5" : Bool;
            "Q2.6" : Bool;
            "Q2.7" : Bool;
         END_STRUCT;
         PlcOutputSafety : Struct   // plc output safety
            "Q900.0" : Bool;
            "Q900.1" : Bool;
            "Q900.2" : Bool;
            "Q900.3" : Bool;
            "Q908.0" : Bool;
            "Q908.1" : Bool;
            "Q908.2" : Bool;
            "Q908.3" : Bool;
         END_STRUCT;
         res : Array[1..200] of Byte;
      END_STRUCT;
   END_VAR
BEGIN
END_DATA_BLOCK

DATA_BLOCK "Enc"   // DB323
{ S7_Optimized_Access := 'TRUE' }
// stored: AutoNumber false, IsRetainMemResEnabled true, MemoryReserve 500, RetainMemoryReserve 500
   VAR RETAIN
      "1BCI1" : "TypeEncoder";   // encoder infeed scanner
      "1BCM1" : "TypeEncoder";   // encoder scanner
      "1BCO1" : "TypeEncoder";   // encoder outfeed scanner
      "8B1.B" : "TypeEncoder";   // light barrier measuring distance for the position of the scanner
      "8BC1.T" : "TypeEncoder";   // encoder adjustment top - normal drive
      "8BC1.L" : "TypeEncoder";   // encoder adjustment left - normal drive
      "8BC1.R" : "TypeEncoder";   // encoder adjustment right - normal drive
      "8U1.T" : "TypeEncoder";   // encoder adjustment top - linear drive
      "8U1.L" : "TypeEncoder";   // encoder adjustment left - linear drive
      "8U1.R" : "TypeEncoder";   // encoder adjustment right - linear drive
   END_VAR
BEGIN
   "1BCI1".ref := FALSE;
   "1BCI1".refMode := FALSE;
   "1BCI1".refRun := FALSE;
   "1BCI1".refOk := FALSE;
   "1BCI1".ready := TRUE;
   "1BCI1".posOk := TRUE;
   "1BCI1".notInPos := FALSE;
   "1BCI1".tarMin := TRUE;
   "1BCI1".tarMax := TRUE;
   "1BCI1".min := FALSE;
   "1BCI1".max := FALSE;
   "1BCI1".minTar := TRUE;
   "1BCI1".maxTar := TRUE;
   "1BCI1".sync := FALSE;
   "1BCI1".comOk := TRUE;
   "1BCI1".errOverflow := FALSE;
   "1BCI1".errRunCheck := FALSE;
   "1BCI1".errLim := FALSE;
   "1BCI1".errCom := FALSE;
   "1BCI1".err := FALSE;
   "1BCI1".errOffDel := TRUE;
   "1BCI1".dirUp := FALSE;
   "1BCI1".dirDn := TRUE;
   "1BCI1".errNr := 0;
   "1BCI1".encAct := 0;
   "1BCI1".resetPos := 0.0;
   "1BCI1".calOffset := 0.0;
   "1BCI1".calGain := 0.0005025126;
   "1BCI1".refPos := 0.0;
   "1BCI1".calP1Inc := 0;
   "1BCI1".calP1Mm := 0.0;
   "1BCI1".calP2Inc := 0;
   "1BCI1".calP2Mm := 0.0;
   "1BCI1".limMin := 0.0;
   "1BCI1".limMax := 0.0;
   "1BCI1".tar := 10.0;
   "1BCI1".act := 0.0;
   "1BCI1".offset := 0.0;
   "1BCI1".deltaInc := 0;
   "1BCI1".delta := 11.31196;
   "1BCI1".tarMinPos := 10.0;
   "1BCI1".tarMaxPos := -10.0;
   "1BCI1".minPos := 0.0;
   "1BCI1".maxPos := 0.0;
   "1BCI1".gPos := 0.0;
   "1BCI1".ePos := 0.0;
   "1BCI1".sPos := 0.0;
   "1BCI1".speed := 16#7FBF_FFFF;
   "1BCI1"."name" := WSTRING#'35BC11';
   "1BCI1".description := WSTRING#'Encoder Zuteiler Anschlag - Zubringung';
   "1BCM1".ref := FALSE;
   "1BCM1".refMode := FALSE;
   "1BCM1".refRun := FALSE;
   "1BCM1".refOk := FALSE;
   "1BCM1".ready := FALSE;
   "1BCM1".posOk := TRUE;
   "1BCM1".notInPos := FALSE;
   "1BCM1".tarMin := TRUE;
   "1BCM1".tarMax := TRUE;
   "1BCM1".min := FALSE;
   "1BCM1".max := FALSE;
   "1BCM1".minTar := TRUE;
   "1BCM1".maxTar := TRUE;
   "1BCM1".sync := FALSE;
   "1BCM1".comOk := FALSE;
   "1BCM1".errOverflow := FALSE;
   "1BCM1".errRunCheck := FALSE;
   "1BCM1".errLim := TRUE;
   "1BCM1".errCom := TRUE;
   "1BCM1".err := FALSE;
   "1BCM1".errOffDel := TRUE;
   "1BCM1".dirUp := FALSE;
   "1BCM1".dirDn := FALSE;
   "1BCM1".errNr := 112;
   "1BCM1".encAct := 0;
   "1BCM1".resetPos := 0.0;
   "1BCM1".calOffset := 0.0;
   "1BCM1".calGain := 0.0;
   "1BCM1".refPos := 0.0;
   "1BCM1".calP1Inc := 0;
   "1BCM1".calP1Mm := 0.0;
   "1BCM1".calP2Inc := 0;
   "1BCM1".calP2Mm := 0.0;
   "1BCM1".limMin := -50.0;
   "1BCM1".limMax := 50.0;
   "1BCM1".tar := 10.0;
   "1BCM1".act := 0.0;
   "1BCM1".offset := 0.0;
   "1BCM1".deltaInc := 0;
   "1BCM1".delta := 11.31196;
   "1BCM1".tarMinPos := 10.0;
   "1BCM1".tarMaxPos := -10.0;
   "1BCM1".minPos := 0.0;
   "1BCM1".maxPos := 0.0;
   "1BCM1".gPos := 0.0;
   "1BCM1".ePos := 0.0;
   "1BCM1".sPos := 0.0;
   "1BCM1".speed := 0.0;
   "1BCM1"."name" := WSTRING#'35BC11';
   "1BCM1".description := WSTRING#'Encoder Zuteiler Anschlag - Zubringung';
   "1BCO1".ref := FALSE;
   "1BCO1".refMode := FALSE;
   "1BCO1".refRun := FALSE;
   "1BCO1".refOk := FALSE;
   "1BCO1".ready := FALSE;
   "1BCO1".posOk := TRUE;
   "1BCO1".notInPos := FALSE;
   "1BCO1".tarMin := TRUE;
   "1BCO1".tarMax := TRUE;
   "1BCO1".min := FALSE;
   "1BCO1".max := FALSE;
   "1BCO1".minTar := TRUE;
   "1BCO1".maxTar := TRUE;
   "1BCO1".sync := FALSE;
   "1BCO1".comOk := FALSE;
   "1BCO1".errOverflow := FALSE;
   "1BCO1".errRunCheck := FALSE;
   "1BCO1".errLim := TRUE;
   "1BCO1".errCom := TRUE;
   "1BCO1".err := FALSE;
   "1BCO1".errOffDel := TRUE;
   "1BCO1".dirUp := FALSE;
   "1BCO1".dirDn := FALSE;
   "1BCO1".errNr := 112;
   "1BCO1".encAct := 0;
   "1BCO1".resetPos := 0.0;
   "1BCO1".calOffset := 0.0;
   "1BCO1".calGain := 0.0;
   "1BCO1".refPos := 0.0;
   "1BCO1".calP1Inc := 0;
   "1BCO1".calP1Mm := 0.0;
   "1BCO1".calP2Inc := 0;
   "1BCO1".calP2Mm := 0.0;
   "1BCO1".limMin := -50.0;
   "1BCO1".limMax := 50.0;
   "1BCO1".tar := 10.0;
   "1BCO1".act := 0.0;
   "1BCO1".offset := 0.0;
   "1BCO1".deltaInc := 0;
   "1BCO1".delta := 11.31196;
   "1BCO1".tarMinPos := 10.0;
   "1BCO1".tarMaxPos := -10.0;
   "1BCO1".minPos := 0.0;
   "1BCO1".maxPos := 0.0;
   "1BCO1".gPos := 0.0;
   "1BCO1".ePos := 0.0;
   "1BCO1".sPos := 0.0;
   "1BCO1".speed := 0.0;
   "1BCO1"."name" := WSTRING#'35BC11';
   "1BCO1".description := WSTRING#'Encoder Zuteiler Anschlag - Zubringung';
   "8B1.B".ref := FALSE;
   "8B1.B".refMode := FALSE;
   "8B1.B".refRun := FALSE;
   "8B1.B".refOk := TRUE;
   "8B1.B".ready := FALSE;
   "8B1.B".posOk := FALSE;
   "8B1.B".notInPos := FALSE;
   "8B1.B".tarMin := FALSE;
   "8B1.B".tarMax := FALSE;
   "8B1.B".min := FALSE;
   "8B1.B".max := FALSE;
   "8B1.B".minTar := FALSE;
   "8B1.B".maxTar := FALSE;
   "8B1.B".sync := FALSE;
   "8B1.B".comOk := FALSE;
   "8B1.B".errOverflow := FALSE;
   "8B1.B".errRunCheck := FALSE;
   "8B1.B".errLim := FALSE;
   "8B1.B".errCom := FALSE;
   "8B1.B".err := FALSE;
   "8B1.B".errOffDel := FALSE;
   "8B1.B".dirUp := FALSE;
   "8B1.B".dirDn := FALSE;
   "8B1.B".errNr := 0;
   "8B1.B".encAct := -2360;
   "8B1.B".resetPos := 0.0;
   "8B1.B".calOffset := 0.0;
   "8B1.B".calGain := 1.0;
   "8B1.B".refPos := 0.0;
   "8B1.B".calP1Inc := 0;
   "8B1.B".calP1Mm := 0.0;
   "8B1.B".calP2Inc := 0;
   "8B1.B".calP2Mm := 0.0;
   "8B1.B".limMin := -505.0;
   "8B1.B".limMax := 505.0;
   "8B1.B".tar := 60.0;
   "8B1.B".act := -236.0;
   "8B1.B".offset := 0.0;
   "8B1.B".deltaInc := 0;
   "8B1.B".delta := 0.0;
   "8B1.B".tarMinPos := -500.0;
   "8B1.B".tarMaxPos := 500.0;
   "8B1.B".minPos := -500.0;
   "8B1.B".maxPos := 500.0;
   "8B1.B".gPos := 0.0;
   "8B1.B".ePos := 0.0;
   "8B1.B".sPos := 0.0;
   "8B1.B".speed := 0.0;
   "8B1.B"."name" := WSTRING#'';
   "8B1.B".description := WSTRING#'';
   "8BC1.T".ref := FALSE;
   "8BC1.T".refMode := TRUE;
   "8BC1.T".refRun := FALSE;
   "8BC1.T".refOk := TRUE;
   "8BC1.T".ready := TRUE;
   "8BC1.T".posOk := FALSE;
   "8BC1.T".notInPos := FALSE;
   "8BC1.T".tarMin := FALSE;
   "8BC1.T".tarMax := FALSE;
   "8BC1.T".min := FALSE;
   "8BC1.T".max := FALSE;
   "8BC1.T".minTar := TRUE;
   "8BC1.T".maxTar := FALSE;
   "8BC1.T".sync := FALSE;
   "8BC1.T".comOk := TRUE;
   "8BC1.T".errOverflow := FALSE;
   "8BC1.T".errRunCheck := FALSE;
   "8BC1.T".errLim := TRUE;
   "8BC1.T".errCom := FALSE;
   "8BC1.T".err := TRUE;
   "8BC1.T".errOffDel := TRUE;
   "8BC1.T".dirUp := TRUE;
   "8BC1.T".dirDn := FALSE;
   "8BC1.T".errNr := 1;
   "8BC1.T".encAct := 1563;
   "8BC1.T".resetPos := 52.98273;
   "8BC1.T".calOffset := 0.0;
   "8BC1.T".calGain := -0.0275;
   "8BC1.T".refPos := 10.0;
   "8BC1.T".calP1Inc := 0;
   "8BC1.T".calP1Mm := 0.0;
   "8BC1.T".calP2Inc := 0;
   "8BC1.T".calP2Mm := 0.0;
   "8BC1.T".limMin := 5.0;
   "8BC1.T".limMax := 215.0;
   "8BC1.T".tar := 12.0;
   "8BC1.T".act := -32.98265;
   "8BC1.T".offset := 0.0;
   "8BC1.T".deltaInc := 0;
   "8BC1.T".delta := 0.0;
   "8BC1.T".tarMinPos := 10.0;
   "8BC1.T".tarMaxPos := 210.0;
   "8BC1.T".minPos := 10.0;
   "8BC1.T".maxPos := 210.0;
   "8BC1.T".gPos := 0.0;
   "8BC1.T".ePos := 0.0;
   "8BC1.T".sPos := 0.0;
   "8BC1.T".speed := 16#7FBF_FFFF;
   "8BC1.T"."name" := WSTRING#'35BC11';
   "8BC1.T".description := WSTRING#'Encoder Zuteiler Anschlag - Zubringung';
   "8BC1.L".ref := FALSE;
   "8BC1.L".refMode := TRUE;
   "8BC1.L".refRun := FALSE;
   "8BC1.L".refOk := TRUE;
   "8BC1.L".ready := TRUE;
   "8BC1.L".posOk := TRUE;
   "8BC1.L".notInPos := FALSE;
   "8BC1.L".tarMin := FALSE;
   "8BC1.L".tarMax := FALSE;
   "8BC1.L".min := FALSE;
   "8BC1.L".max := FALSE;
   "8BC1.L".minTar := FALSE;
   "8BC1.L".maxTar := FALSE;
   "8BC1.L".sync := FALSE;
   "8BC1.L".comOk := TRUE;
   "8BC1.L".errOverflow := FALSE;
   "8BC1.L".errRunCheck := FALSE;
   "8BC1.L".errLim := FALSE;
   "8BC1.L".errCom := FALSE;
   "8BC1.L".err := FALSE;
   "8BC1.L".errOffDel := FALSE;
   "8BC1.L".dirUp := TRUE;
   "8BC1.L".dirDn := FALSE;
   "8BC1.L".errNr := 0;
   "8BC1.L".encAct := 638;
   "8BC1.L".resetPos := 9.972851;
   "8BC1.L".calOffset := 0.0;
   "8BC1.L".calGain := -0.0275;
   "8BC1.L".refPos := 10.0;
   "8BC1.L".calP1Inc := 0;
   "8BC1.L".calP1Mm := 0.0;
   "8BC1.L".calP2Inc := 0;
   "8BC1.L".calP2Mm := 0.0;
   "8BC1.L".limMin := 5.0;
   "8BC1.L".limMax := 215.0;
   "8BC1.L".tar := 87.5;
   "8BC1.L".act := 87.52025;
   "8BC1.L".offset := 0.0;
   "8BC1.L".deltaInc := 0;
   "8BC1.L".delta := 0.0;
   "8BC1.L".tarMinPos := 10.0;
   "8BC1.L".tarMaxPos := 210.0;
   "8BC1.L".minPos := 10.0;
   "8BC1.L".maxPos := 210.0;
   "8BC1.L".gPos := 0.0;
   "8BC1.L".ePos := 0.0;
   "8BC1.L".sPos := 0.0;
   "8BC1.L".speed := 16#7FBF_FFFF;
   "8BC1.L"."name" := WSTRING#'35BC11';
   "8BC1.L".description := WSTRING#'Encoder Zuteiler Anschlag - Zubringung';
   "8BC1.R".ref := FALSE;
   "8BC1.R".refMode := TRUE;
   "8BC1.R".refRun := FALSE;
   "8BC1.R".refOk := TRUE;
   "8BC1.R".ready := TRUE;
   "8BC1.R".posOk := TRUE;
   "8BC1.R".notInPos := FALSE;
   "8BC1.R".tarMin := FALSE;
   "8BC1.R".tarMax := FALSE;
   "8BC1.R".min := FALSE;
   "8BC1.R".max := FALSE;
   "8BC1.R".minTar := FALSE;
   "8BC1.R".maxTar := FALSE;
   "8BC1.R".sync := FALSE;
   "8BC1.R".comOk := TRUE;
   "8BC1.R".errOverflow := FALSE;
   "8BC1.R".errRunCheck := FALSE;
   "8BC1.R".errLim := FALSE;
   "8BC1.R".errCom := FALSE;
   "8BC1.R".err := FALSE;
   "8BC1.R".errOffDel := FALSE;
   "8BC1.R".dirUp := TRUE;
   "8BC1.R".dirDn := FALSE;
   "8BC1.R".errNr := 0;
   "8BC1.R".encAct := 636;
   "8BC1.R".resetPos := 10.00027;
   "8BC1.R".calOffset := 0.0;
   "8BC1.R".calGain := -0.0275;
   "8BC1.R".refPos := 10.0;
   "8BC1.R".calP1Inc := 0;
   "8BC1.R".calP1Mm := 0.0;
   "8BC1.R".calP2Inc := 0;
   "8BC1.R".calP2Mm := 0.0;
   "8BC1.R".limMin := 5.0;
   "8BC1.R".limMax := 215.0;
   "8BC1.R".tar := 82.6;
   "8BC1.R".act := 82.62568;
   "8BC1.R".offset := 0.0;
   "8BC1.R".deltaInc := 0;
   "8BC1.R".delta := 0.0;
   "8BC1.R".tarMinPos := 10.0;
   "8BC1.R".tarMaxPos := 210.0;
   "8BC1.R".minPos := 10.0;
   "8BC1.R".maxPos := 210.0;
   "8BC1.R".gPos := 0.0;
   "8BC1.R".ePos := 0.0;
   "8BC1.R".sPos := 0.0;
   "8BC1.R".speed := 16#7FBF_FFFF;
   "8BC1.R"."name" := WSTRING#'35BC11';
   "8BC1.R".description := WSTRING#'Encoder Zuteiler Anschlag - Zubringung';
   "8U1.T".ref := TRUE;
   "8U1.T".refMode := TRUE;
   "8U1.T".refRun := FALSE;
   "8U1.T".refOk := FALSE;
   "8U1.T".ready := FALSE;
   "8U1.T".posOk := FALSE;
   "8U1.T".notInPos := FALSE;
   "8U1.T".tarMin := TRUE;
   "8U1.T".tarMax := TRUE;
   "8U1.T".min := FALSE;
   "8U1.T".max := FALSE;
   "8U1.T".minTar := TRUE;
   "8U1.T".maxTar := TRUE;
   "8U1.T".sync := FALSE;
   "8U1.T".comOk := FALSE;
   "8U1.T".errOverflow := FALSE;
   "8U1.T".errRunCheck := FALSE;
   "8U1.T".errLim := TRUE;
   "8U1.T".errCom := TRUE;
   "8U1.T".err := FALSE;
   "8U1.T".errOffDel := TRUE;
   "8U1.T".dirUp := FALSE;
   "8U1.T".dirDn := FALSE;
   "8U1.T".errNr := 112;
   "8U1.T".encAct := 0;
   "8U1.T".resetPos := 0.0;
   "8U1.T".calOffset := 0.0;
   "8U1.T".calGain := 1.0;
   "8U1.T".refPos := 0.0;
   "8U1.T".calP1Inc := 0;
   "8U1.T".calP1Mm := 0.0;
   "8U1.T".calP2Inc := 0;
   "8U1.T".calP2Mm := 0.0;
   "8U1.T".limMin := -5.0;
   "8U1.T".limMax := 155.0;
   "8U1.T".tar := 42.0;
   "8U1.T".act := 0.0;
   "8U1.T".offset := 0.0;
   "8U1.T".deltaInc := 0;
   "8U1.T".delta := 0.0;
   "8U1.T".tarMinPos := 0.0;
   "8U1.T".tarMaxPos := 150.0;
   "8U1.T".minPos := 0.0;
   "8U1.T".maxPos := 150.0;
   "8U1.T".gPos := 0.0;
   "8U1.T".ePos := 0.0;
   "8U1.T".sPos := 0.0;
   "8U1.T".speed := 0.0;
   "8U1.T"."name" := WSTRING#'35BC11';
   "8U1.T".description := WSTRING#'Encoder Zuteiler Anschlag - Zubringung';
   "8U1.L".ref := TRUE;
   "8U1.L".refMode := TRUE;
   "8U1.L".refRun := FALSE;
   "8U1.L".refOk := FALSE;
   "8U1.L".ready := FALSE;
   "8U1.L".posOk := FALSE;
   "8U1.L".notInPos := FALSE;
   "8U1.L".tarMin := TRUE;
   "8U1.L".tarMax := TRUE;
   "8U1.L".min := FALSE;
   "8U1.L".max := FALSE;
   "8U1.L".minTar := TRUE;
   "8U1.L".maxTar := TRUE;
   "8U1.L".sync := FALSE;
   "8U1.L".comOk := FALSE;
   "8U1.L".errOverflow := FALSE;
   "8U1.L".errRunCheck := FALSE;
   "8U1.L".errLim := TRUE;
   "8U1.L".errCom := TRUE;
   "8U1.L".err := FALSE;
   "8U1.L".errOffDel := TRUE;
   "8U1.L".dirUp := FALSE;
   "8U1.L".dirDn := FALSE;
   "8U1.L".errNr := 112;
   "8U1.L".encAct := 0;
   "8U1.L".resetPos := 0.0;
   "8U1.L".calOffset := 0.0;
   "8U1.L".calGain := 1.0;
   "8U1.L".refPos := 0.0;
   "8U1.L".calP1Inc := 0;
   "8U1.L".calP1Mm := 0.0;
   "8U1.L".calP2Inc := 0;
   "8U1.L".calP2Mm := 0.0;
   "8U1.L".limMin := -5.0;
   "8U1.L".limMax := 155.0;
   "8U1.L".tar := 82.5;
   "8U1.L".act := 0.0;
   "8U1.L".offset := 0.0;
   "8U1.L".deltaInc := 0;
   "8U1.L".delta := 0.0;
   "8U1.L".tarMinPos := 0.0;
   "8U1.L".tarMaxPos := 150.0;
   "8U1.L".minPos := 0.0;
   "8U1.L".maxPos := 150.0;
   "8U1.L".gPos := 0.0;
   "8U1.L".ePos := 0.0;
   "8U1.L".sPos := 0.0;
   "8U1.L".speed := 0.0;
   "8U1.L"."name" := WSTRING#'35BC11';
   "8U1.L".description := WSTRING#'Encoder Zuteiler Anschlag - Zubringung';
   "8U1.R".ref := TRUE;
   "8U1.R".refMode := TRUE;
   "8U1.R".refRun := FALSE;
   "8U1.R".refOk := FALSE;
   "8U1.R".ready := FALSE;
   "8U1.R".posOk := FALSE;
   "8U1.R".notInPos := FALSE;
   "8U1.R".tarMin := TRUE;
   "8U1.R".tarMax := TRUE;
   "8U1.R".min := FALSE;
   "8U1.R".max := FALSE;
   "8U1.R".minTar := TRUE;
   "8U1.R".maxTar := TRUE;
   "8U1.R".sync := FALSE;
   "8U1.R".comOk := FALSE;
   "8U1.R".errOverflow := FALSE;
   "8U1.R".errRunCheck := FALSE;
   "8U1.R".errLim := TRUE;
   "8U1.R".errCom := TRUE;
   "8U1.R".err := FALSE;
   "8U1.R".errOffDel := TRUE;
   "8U1.R".dirUp := FALSE;
   "8U1.R".dirDn := FALSE;
   "8U1.R".errNr := 112;
   "8U1.R".encAct := 0;
   "8U1.R".resetPos := 0.0;
   "8U1.R".calOffset := 0.0;
   "8U1.R".calGain := 1.0;
   "8U1.R".refPos := 0.0;
   "8U1.R".calP1Inc := 0;
   "8U1.R".calP1Mm := 0.0;
   "8U1.R".calP2Inc := 0;
   "8U1.R".calP2Mm := 0.0;
   "8U1.R".limMin := -5.0;
   "8U1.R".limMax := 155.0;
   "8U1.R".tar := 82.5;
   "8U1.R".act := 0.0;
   "8U1.R".offset := 0.0;
   "8U1.R".deltaInc := 0;
   "8U1.R".delta := 0.0;
   "8U1.R".tarMinPos := 0.0;
   "8U1.R".tarMaxPos := 150.0;
   "8U1.R".minPos := 0.0;
   "8U1.R".maxPos := 150.0;
   "8U1.R".gPos := 0.0;
   "8U1.R".ePos := 0.0;
   "8U1.R".sPos := 0.0;
   "8U1.R".speed := 0.0;
   "8U1.R"."name" := WSTRING#'35BC11';
   "8U1.R".description := WSTRING#'Encoder Zuteiler Anschlag - Zubringung';
END_DATA_BLOCK

